// TIA Portal V21 export
DATA_BLOCK "DB610"   // DB610
TITLE = DB610
AUTHOR : PRECISE
FAMILY : PRECISE
// CIP SYSTEM DRAIN
// stored: AutoNumber false, InstanceOfName FB610, InstanceOfType FB
"FB610"
   // VAR_INPUT
   //    CycleEnable : Bool;
   //    CycleRunning : Bool;
   //    SecPulse : Bool;
   //    AlwaysTrue : Bool;
   //    SetTime : Int;
   //    Loops : Int;
   //    DelayBetweenLoops : Int;
   // END_VAR
   // VAR_OUTPUT
   //    Started : Bool;
   //    ParaOut : "SystemDrainOutputs";
   //    TimePv : DInt;
   //    StepStatus : String[60];
   // END_VAR
   // VAR_IN_OUT
   //    Over : Bool;
   //    OverTemp : Bool;
   //    Popup : Bool;
   //    PopupAck : Bool;
   //    PopUpSel : Bool;
   // END_VAR
   // VAR
   //    RE1 : Bool;
   //    "Timer" { S7_SetPoint := 'True'} : "FB101";
   // END_VAR
BEGIN
END_DATA_BLOCK
